FUNCTION_BLOCK LOADING_PICKLE
  {SET_ATTRIBUTE(OpcUa, SERVICE)}
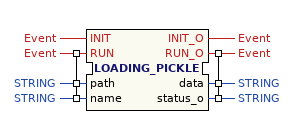
  EVENT_INPUT
    INIT;
    RUN WITH path, name; {SET_ATTRIBUTE(OpcUa, Method)}
  END_EVENT
  EVENT_OUTPUT
    INIT_O;
    RUN_O WITH data, status_o;
  END_EVENT
  VAR_INPUT
    path : STRING; {SET_ATTRIBUTE(OpcUa, Variable.RUN)}
    name : STRING; {SET_ATTRIBUTE(OpcUa, Variable.RUN)}
  END_VAR
  VAR_OUTPUT
    data : STRING; {SET_ATTRIBUTE(OpcUa, Variable.RUN)}
    status_o : STRING; {SET_ATTRIBUTE(OpcUa, Variable.RUN)}
  END_VAR
END_FUNCTION_BLOCK
